// TIA Portal V19 export
FUNCTION_BLOCK "LAF_InterfaceSignalsBool"   // FB52, LAD
TITLE = LAF_InterfaceSignalsBool / Schnittstelle für boolsche Signale
AUTHOR : Siemens Digital Industries
FAMILY : LAF
VERSION : 1.2
// The block cyclically evaluates the status of the configured Boolean signals and transfers the values to the configured data (HMI) interface. The symbolic name of the configured tags will be read once only, triggered by the selection of a signal dataset on the HMI, and will be transferred to the HMI interface as well.  
// The block and the associated WinCC screen are designed for 16 signal datasets with 32 signals each  (“Page 1” through “Page 16”).  The signal dataset can be selected in the WinCC-screen.  
// 
// * The maximum length of the symbol name is limited to 40 characters.  
// 
// For further notes see:  [CallInterfaceSignals](../Function%20Blocks/CallInterfaceSignals.htm)  
// 
// **PLC Data types**  
// * LAF_typeInterfaceSignals  
// + LAF_typeInterfaceSignalsBool  
// 
// **WinCC Screen**  
// {.pageWidth}
// ![Image](LAF_InterfaceSignalsBool/en/image1.PNG)
// 
// **Block call example**  
// {.pageWidth}
// ![Image](LAF_InterfaceSignalsBool/en/image4.PNG)
// View in ladder logic (LAD).  
// 
// **Calling Interface**  
// The block has to be called in the cyclic program in “CallInterfaceSignals”.  
// The block handles 16 Boolean signals. Since one HMI screen can display 32 signals, it is necessary to call the block two times.  
// 
// **Internally used “Extended instructions / blocks“**  
// GetSymbolName
// Die hier aufgeführten Bausteine gehören zum mehrsprachigen Alarm-Bausteinpaket von SICAR in Verbindung mit dem Softwarepaket „ProDiag“.  
// Alle Bausteine besitzt mehrere Input-Parameter „….TriggerX“ an die ein oder mehrere logische Verknüpfungen angelegt werden können. Die Trigger-Eingänge werden mittels ProDiag auf eine Operanden Überwachung überwacht (“Eigenschaften > Überwachung > Allgemein > Überwachungsart: Operand“). Demzufolge sind sie im Fehlerfall auch über den PLC-Code-Viewer auf dem HMI diagnostizierbar.  
// Entsprechend den Überwachungseinstellungen von „ProDiag“ werden die Meldetexte gebildet und erscheinen auf dem HMI in der Meldeanzeige (Bilder: „Meldungen“ / „Alarms“ und „Meldearchiv“ / „Alarms history“). Die Bausteine greifen dazu auf Texte von PLC-Meldetextlisten zu. 
// Eine Meldung kann mehrsprachig ausgeführt werden. Bereits ausgeführte Sprachen sind Englisch und Deutsch; weitere Sprachen sind frei wählbar.  
// Die auf dem HMI angezeigte Sprachvariante wird im Bild „System & Einstellungen“ / “System & Settings“ mit den Buttons der Länderflaggen ausgewählt. Das Bild ist erreichbar, über den Button „System“ (unten rechts im Bild).  
// Ein Bausteinaufruf kann max. 16 Meldungen bearbeiten.  
// 
// WARNING 
// :     Innerhalb des Bausteins wird aufgrund der ProDiag-Überwachung auf PLC-Meldetextliste „GLOBAL_GENERAL_AlarmTextList“ und deren Einträge fest verwiesen. 
// :     ![Icon](_Icon/prohibition.PNG) {.alignLeft} Ändern Sie nicht den Namen dieser PLC-Meldetextliste; der Name wird bei einem Übersetzen im Baustein nicht automatisch nachgeführt!
// :     ![Icon](_Icon/prohibition.PNG) {.alignLeft} Ändern Sie nicht die Reihenfolge der Einträge in der bereits existierenden PLC-Meldetextliste. Diese werden fest referenziert! 
// :     ![Icon](_Icon/information.PNG) {.alignLeft} Sie können stattdessen einen Eintrag in der PLC-Meldetextliste neu hinzufügen.  
// 
// ---
// 
// NOTE
// :     Beachten Sie dabei bitte, dass bei SICAR-Versionsänderungen auch Einträge in den PLC-Meldetextlisten geändert/hinzugefügt werden können, aufgrund dessen es dann zu Doppelbelegungen kommen kann. 
// :     Es ist daher sinnvoll weitere „USER…“-Textliste(n) zu erstellen, losgelöst von den in SICAR bereits existierenden PLC-Meldetextlisten 
// 
// ---
// 
// Es sind folgende Bausteine verfügbar: 
// 
// * LSicar_AlarmOp16_PrD: 		16 Operanden Alarme (rote Hintergrundfarbe im Alarm-Bild)
// * LSicar_WarnOp16_PrD: 		16 Operanden Warnungen (orange Hintergrundfarbe im Alarm-Bild) 
// * LSicar_InfoOp16_PrD: 		16 Operanden Informationen (blaue Hintergrundfarbe im Alarm-Bild) 
// *  LSicar_AlarmOpFsafe8_PrD: 		8 Operanden F-Alarme (gelbe Hintergrundfarbe im Alarm-Bild) 
// 
// **Überwachungsart**  
// 
// ![Image](LSicar_AlarmOp16_PrD/de/image1.PNG) 
// 
// Der Text für die Überwachungsart „Fehlermeldung“ ist in den  Überwachungseinstellungen „Allgemein > Überwachungsart > Eigenschaften“ mit -Op- angegeben und bei der Projektierung der „Meldetexte > FB-Parameter“ im Meldetext konfiguriert.  
// 
// **_AlarmOp16_PrD**  
// In den ProDiag-Überwachungseinstellungen ist die Kategorie: „Alarm“ definiert und wird für alle Inputs verwendet. Dieser Kategorie ist die Meldeklasse „ Alarm_ProDiag“ zugeordnet. Auf dem HMI ist dieser Meldeklasse unter „HMI-Meldungen > Lasche ‚Meldeklasse‘“ die Hintergrundfarbe Rot zugeordnet mit dem Anzeigename „Alarm“. Somit erscheinen Meldungen im Alarm-Bild wie folgt (Beispiel):  
// 
// ![Image](LSicar_AlarmOp16_PrD/de/image2.PNG)  
// 
// Zudem werden die Alarme auf eine Statische Variable „HMI_Alarm“ kopiert. Diese kann dazu benutzt werden um ein HMI-Variable zu generieren und -somit auf dem HMI- die Signale zu Animationszwecken zu nutzen.  
// 
// **_WarnOp16_PrD**  
// In den ProDiag-Überwachungseinstellungen ist die Kategorie: „Warn“ definiert und wird für alle Inputs verwendet. Dieser Kategorie ist die Meldeklasse „ Warning_ProDiag“ zugeordnet. Auf dem HMI ist dieser Meldeklasse unter „HMI-Meldungen > Lasche ‚Meldeklasse‘“ die Hintergrundfarbe Orange zugeordnet mit dem Anzeigename „Warn“. Somit erscheinen Meldungen im Alarm-Bild wie folgt (Beispiel):  
// 
// ![Image](LSicar_AlarmOp16_PrD/de/image3.PNG)
// 
// The warnings are also copied to a static tag “HMI_Warn”. This can be used to generate a HMI tag, e.g. to use the signals for animations on the HMI.  
// 
// **_InfoOp16_PrD**  
// In den ProDiag-Überwachungseinstellungen ist die Kategorie: „Info“ definiert und wird für alle Inputs verwendet. Dieser Kategorie ist die Meldeklasse „ Information_ProDiag“ zugeordnet. Auf dem HMI ist dieser Meldeklasse unter „HMI-Meldungen > Lasche ‚Meldeklasse‘“ die Hintergrundfarbe Blau zugeordnet mit dem Anzeigename „Info“. Somit erscheinen Meldungen im Alarm-Bild wie folgt (Beispiel):  
// 
// ![Image](LSicar_AlarmOp16_PrD/de/image4.PNG)
// 
// Zudem werden die Warnungen auf eine Statische Variable „HMI_Warn“ kopiert. Diese kann dazu benutzt werden um ein HMI-Variable zu generieren und -somit auf dem HMI- die Signale zu Animationszwecken zu nutzen.  
// 
// **_AlarmOpFsafe8_PrD**  
// In den ProDiag-Überwachungseinstellungen ist die Kategorie: „F-Alarm“ definiert und wird für alle Inputs verwendet. Dieser Kategorie ist die Meldeklasse „F-Alarm_ProDiag“ zugeordnet. Auf dem HMI ist dieser Meldeklasse unter „HMI-Meldungen > Lasche ‚Meldeklasse‘“ die Hintergrundfarbe Gelb zugeordnet mit dem Anzeigename „F-Alarm“. Somit erscheinen Meldungen im Alarm-Bild wie folgt (Beispiel):  
// 
// ![Image](LSicar_AlarmOp16_PrD/de/image5.PNG)
// 
// Zudem werden die Meldungen auf Statische Variablen „HMI_Alarm…“ kopiert. Diese können dazu benutzt werden um HMI-Variablen zu generieren und -somit auf dem HMI- die Signale zu Animationszwecken zu nutzen.  
// 
//  
// #### ProDiag-Meldung in 3 Schritten 
// 
// {.pageWidth}
// ![Image](LSicar_AlarmOp16_PrD/de/image6.PNG)
// 
// **1) Legen Sie eine PLC-Meldetextliste an**
// 1. Öffnen Sie dazu (im Projektbaum) „PLC-Meldetextlisten“ und vergeben Sie einen Namen, hier „Demo_Alarm_PD“.  
// 2. Geben Sie den jeweiligen Meldetext in die Spalte „Eintrag“ ein.
// 	- Achten Sie darauf das die Spalten „Bereich von“ und „Bereich bis“ den gleichen Wert haben.  
// 	- Beginnen Sie mit dem Wert 1.  
// 	- Der Eintrag 1 entspricht dem FB-Parameter „…_trigger1“,  
// 	- Eintrag 2 entspricht FB-Parameter „…_trigger2“, usw.  
// 
// 3. Projektieren Sie die Einträge in den gewünschten Sprachen (hier: Deutsch und Englisch). 
// 
// {.pageWidth}
// ![Image](LSicar_AlarmOp16_PrD/de/image7.PNG)
// 
// **2) Eintrag in „GLOBAL_GENERAL_AlarmTextList“**  
// 1. Öffnen Sie die Textliste „GLOBAL_GENERAL_AlarmTextList“.  
// 2. Tragen Sie den Namen der Textliste, die Sie erzeugt haben, als einen neuen Eintrag ein. Fügen Sie sie dabei als neuen Eintrag hinzu (hier Eintrag 25). Geben Sie dabei den Namen der Textliste als Begleitwert ein mit @4%t#<Namen>@.  
// 3. Projektieren Sie dies in allen gewünschten Sprachen.  
//  
// {.pageWidth}
// ![Image](LSicar_AlarmOp16_PrD/de/image8.PNG)
//  
// **3 Rufen Sie den Alarm-Baustein auf**   
// 1. Geben Sie beim Parameter „plantIdentifier“ einen zusätzlichen Text an. Dieser erscheint ebenso im Meldetext.  
// 2. Beim Parameter „globalAlarmTextlistItem“ geben Sie den Wert des Eintrags an „Bereich von“ / „Bereich bis“, unter dem Ihre Textliste in der „GLOBAL_GENERAL_AlarmTextList“ eingetragen ist, hier 25; damit verweisen Sie auf Ihre PLC-Meldetextliste.  
// 3. Versorgen Sie die Trigger-Eingänge.  
// 
// {.pageWidth}
// ![Image](LSicar_AlarmOp16_PrD/de/image9.PNG)
// 
// **Ergebnise:**  
// Wechselt der Trigger-Eingang auf „1“-Signal, so erscheint die Meldung im Alarm-Bild (entsprechend der ProDiag-Konfiguration) und es kann in den PLC-Code-Viewer verzweigt werden.  
// 
// {.pageWidth}
// ![Image](LSicar_AlarmOp16_PrD/de/image10.PNG)
// 
// 
// **Beispielaufruf**  
// Abbildung in Kontaktplan (KOP), ohne Parameterbeschaltung.  
// Ein lauffähiger Programm-Aufruf hierzu ist im „SICAR-StartUp“-Projekt enthalten.  
// 
// **Aufrufschnittstelle**
// Der Baustein wird im zyklischen Programm aufgerufen.
// stored: Access Published, IsIECCheckEnabled true, MemoryReserve 100, SetENOAutomatically true
   VAR_INPUT
      signal00 { ExternalAccessible := 'False'; ExternalVisible := 'False'; ExternalWritable := 'False'} : Bool;   // Boolesches Signal (01) dessen Status und symbolischer Name am HMI dargestellt werden soll. Hinweis: Der symbolische Namen wird mit max. 32 Zeichen darge-stellt. / Boolean signal (number 01) to be displayed on the HMI with status and symbolic name.
      signal01 { ExternalAccessible := 'False'; ExternalVisible := 'False'; ExternalWritable := 'False'} : Bool;   // Analoge Parametrierung wie bei Input „signal01“ / Similar configuration as for “signal01“
      signal02 { ExternalAccessible := 'False'; ExternalVisible := 'False'; ExternalWritable := 'False'} : Bool;   // Analoge Parametrierung wie bei Input „signal01“ / Similar configuration as for “signal01“
      signal03 { ExternalAccessible := 'False'; ExternalVisible := 'False'; ExternalWritable := 'False'} : Bool;   // Analoge Parametrierung wie bei Input „signal01“ / Similar configuration as for “signal01“
      signal04 { ExternalAccessible := 'False'; ExternalVisible := 'False'; ExternalWritable := 'False'} : Bool;   // Analoge Parametrierung wie bei Input „signal01“ / Similar configuration as for “signal01“
      signal05 { ExternalAccessible := 'False'; ExternalVisible := 'False'; ExternalWritable := 'False'} : Bool;   // Analoge Parametrierung wie bei Input „signal01“ / Similar configuration as for “signal01“
      signal06 { ExternalAccessible := 'False'; ExternalVisible := 'False'; ExternalWritable := 'False'} : Bool;   // Analoge Parametrierung wie bei Input „signal01“ / Similar configuration as for “signal01“
      signal07 { ExternalAccessible := 'False'; ExternalVisible := 'False'; ExternalWritable := 'False'} : Bool;   // Analoge Parametrierung wie bei Input „signal01“ / Similar configuration as for “signal01“
      signal08 { ExternalAccessible := 'False'; ExternalVisible := 'False'; ExternalWritable := 'False'} : Bool;   // Analoge Parametrierung wie bei Input „signal01“ / Similar configuration as for “signal01“
      signal09 { ExternalAccessible := 'False'; ExternalVisible := 'False'; ExternalWritable := 'False'} : Bool;   // Analoge Parametrierung wie bei Input „signal01“ / Similar configuration as for “signal01“
      signal10 { ExternalAccessible := 'False'; ExternalVisible := 'False'; ExternalWritable := 'False'} : Bool;   // Analoge Parametrierung wie bei Input „signal01“ / Similar configuration as for “signal01“
      signal11 { ExternalAccessible := 'False'; ExternalVisible := 'False'; ExternalWritable := 'False'} : Bool;   // Analoge Parametrierung wie bei Input „signal01“ / Similar configuration as for “signal01“
      signal12 { ExternalAccessible := 'False'; ExternalVisible := 'False'; ExternalWritable := 'False'} : Bool;   // Analoge Parametrierung wie bei Input „signal01“ / Similar configuration as for “signal01“
      signal13 { ExternalAccessible := 'False'; ExternalVisible := 'False'; ExternalWritable := 'False'} : Bool;   // Analoge Parametrierung wie bei Input „signal01“ / Similar configuration as for “signal01“
      signal14 { ExternalAccessible := 'False'; ExternalVisible := 'False'; ExternalWritable := 'False'} : Bool;   // Analoge Parametrierung wie bei Input „signal01“ / Similar configuration as for “signal01“
      signal15 { ExternalAccessible := 'False'; ExternalVisible := 'False'; ExternalWritable := 'False'} : Bool;   // Analoge Parametrierung wie bei Input „signal01“ / Similar configuration as for “signal01“
   END_VAR
   VAR_IN_OUT
      interfaceSignals : "LAF_typeInterfaceSignalsBool";   // Im FB “CallInterfaceSignals“ existiert die Struktur „statInterfaceSignalsHmi“ (Array[0..16] of „typeInterfaceSignals-Hmi“). In jeder Struktur existieren die Elemente: - „valueSymboLeft“ und - „valueSymbolRight“mit dem Datentyp "_typeInterfaceSignalsBool"“. Die Nummer des Arrays entspricht dem Signaldatensatz: - Array [1]: Signaldatensatz 1 - Array [2]: Signaldatensatz 2 - usw.Array Index [0] ist nicht zulässig.Zuweisung der entsprechenden Variablen, wie nachfolgend beispiel-haft dargestellt. Der rechte Aufruf entspricht den 16 Signalen auf der rechten Seite des Bildes, der linke Aufruf der linken Seite. / “CallInterfaceSignals“ contains the structure “statInterfaceSignalsHmi“ (Array[0..16] of „typeInterfaceSignalsHmi“). Within each structure there are the two elements: “valueSymbolLeft” and “valueSymbolRight” of the data type “LAF_typeInterfaceSignalsBool“. The number of the array correlates with the number of the signal data-set: Array [1]: Signal data set 1 and Array [2]: Signal data set 2 etc. Array index [0] is not permitted.
   END_VAR
   VAR_TEMP
      tempDummyBool : Bool;   // Dummy
   END_VAR
BEGIN

REGION Network 1: Header Info / Änderungshistorie
   // SIEMENS AG / (c)Copyright 2024
   // ------------------------------------------------------------------------------
   // Title:            LAF_InterfaceSignalsBool
   // Comment/Function: The block cyclically evaluates the status of the configured Boolean signals and transfers the values to the configured data (HMI) interface.
   // Library/Family:           Library of Automation Framework
   // Author:             Siemens Digital Industry
   // Tested with:    S7-PLCSIM Advanced 6.0
   // Engineering:   TIA Portal V19
   // Restrictions:     ---
   // Requirements: ---
   // ------------------------------------------------------------------------------
   // Change log table:
   // Version | Date | Expert in charge | Changes applied
   // -------|---------|-------------|--------------------------------------------
   // 01.02.00 | 30.09.2024 | SIMATIC Systems Support | First released version
   // Die Änderungshistorie wird nur in englischer Editiersprache geführt.
END_REGION

REGION Network 2: Description / Beschreibung
   // **Operation mode Automatic / Manual**  
   // The block is independent of the operation modes and is not assigned to any operation mode area.  
   // 
   // **Alarms**  
   // The block does not generate alarms.  
   // 
   // #### PLC Data types  
   // 
   // The PLC data types are used to structure the data in FB “CallInterfaceSignals“.  
   // 
   // * [LAF_typeInterfaceSignals](../Library%20Types/LAF_typeInterfaceSignals.htm)  
   // * [LAF_typeInterfaceSignalsBool](../Library%20Types/LAF_typeInterfaceSignalsBool.htm)  
   // 
   // #### WinCC-Screen objects 
   // 
   // **WinCC Diagnostic screen**  
   // The screen is located in the project in HMI part under screens -> 09_Diagnostics.  
   // The selection of the interface signal screens is done via the navigation screens which are stored in 00_Screenlayout -> ThirdMenus.  
   // The status is animated in terms of color. Status TRUE = green, Status FALSE = gray.  
   // 
   // **Example**  
   // The Boolean status of the system and clock bit memories are displayed in the screen. The corresponding dataset can be selected via the third navigation bar on the left side of the screen. A headline text can be 
   // entered for each column in the PLC – InstInterfaceSignals DB -> statInterfaceSignalsHmi.  
   // 
   // {.pageWidth}
   // ![Image](LAF_InterfaceSignalsBool/en/image3.PNG)
   // 
   //  
   // #### Further information 
   // 
   // #### Update info 
   // 
   // #### Further documentation  
   // * See [CallInterfaceSignals](../Function%20Blocks/CallInterfaceSignals.htm)
   // **Betriebsart Automatik/Hand**  
   // Der Baustein ist Betriebsarten unabhängig und wird daher keinem Betriebsartenbereich zugewiesen.  
   // 
   // **Alarme**  
   // Der Baustein löst keine eigenen Alarme aus.  
   // 
   // **Beispiel** 
   // 1)	Der Baustein wird aufgerufen mit globalAlarmTextlistItem:= 1. Damit wird auf die PLC-Meldetextliste „OPMode01_Alarm_PD“ verwiesen. Der Input „alarmTrigger1“ zeigt auf den 1. Eintrag in dieser PLC-Meldetextliste.  
   // 2)	Die Überwachung an „alarmTrigger1“ soll auf „0“-Signal (False) überwacht werden; daher die NOT-Verknüpfung.  
   // 
   // {.pageWidth}
   // ![Image](LSicar_AlarmOp16_PrD/de/image10.PNG)
   // 
   // 3)	Die Meldung wird im Alarmbild dargestellt  
   // 4)	und kann im PLC-Viewer beobachtet werden.  
   // 
   // {.pageWidth}
   // ![Image](LSicar_AlarmOp16_PrD/de/image11.PNG)
   // 
   // #### Weitere Dokumente
   // 
   // ![Icon](_Icon/reference.PNG)  
   // 
   // - ProDiag Einstellungen in SICAR: ..\SICAR_Global\SICAR_ProDiag_Settings.pdf  
   // - SICAR PLC Meldetextlisten: ..\SICAR_Global\SICAR_PLC_AlarmTextLists.pdf
END_REGION

REGION Network 3: Update boolean value / Aktualisieren der boolschen Werte
   // Cyclic update of the boolean signal, if the screen is loaded / Wert des Boolschen Signals wird zyklisch aktualisiert, wenn das Bild aufgerufen ist
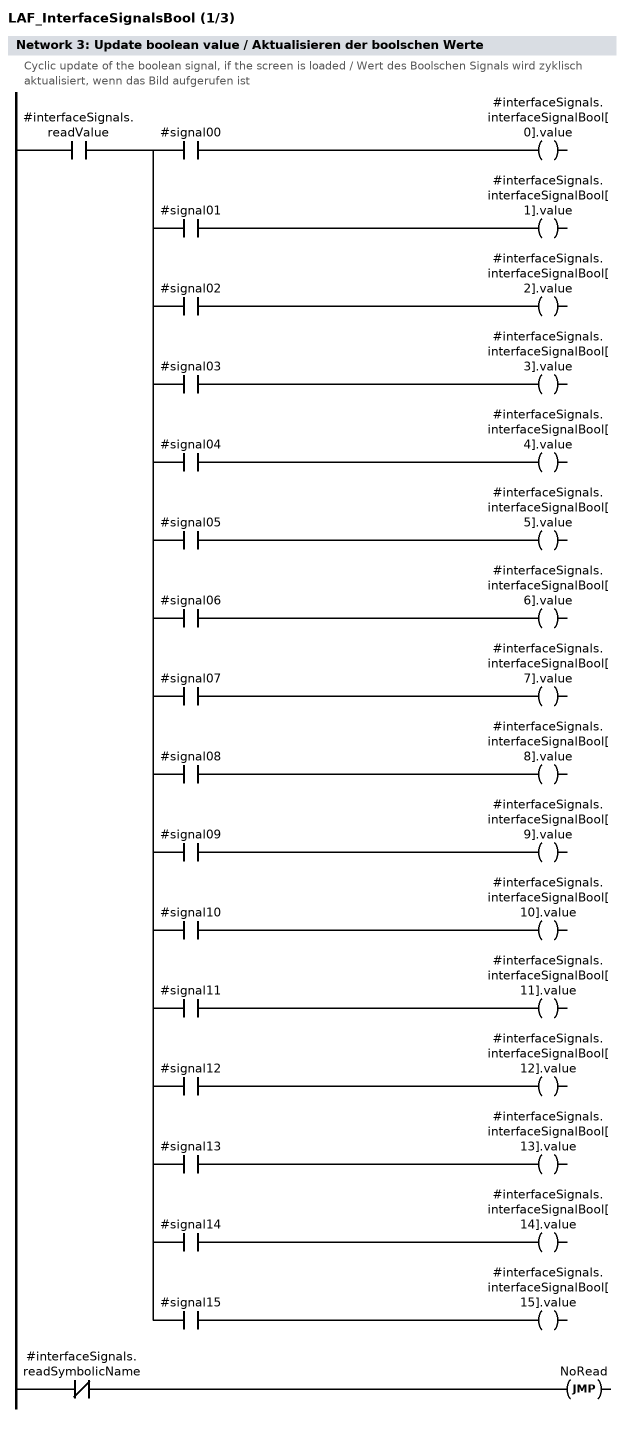
   RUNG wire#powerrail
      Contact( #interfaceSignals.readValue )
      wire#w1
      Contact( #signal00 )
      Coil( #interfaceSignals.interfaceSignalBool[0].value )
   END_RUNG
   RUNG wire#w1
      Contact( #signal01 )
      Coil( #interfaceSignals.interfaceSignalBool[1].value )
   END_RUNG
   RUNG wire#w1
      Contact( #signal02 )
      Coil( #interfaceSignals.interfaceSignalBool[2].value )
   END_RUNG
   RUNG wire#w1
      Contact( #signal03 )
      Coil( #interfaceSignals.interfaceSignalBool[3].value )
   END_RUNG
   RUNG wire#w1
      Contact( #signal04 )
      Coil( #interfaceSignals.interfaceSignalBool[4].value )
   END_RUNG
   RUNG wire#w1
      Contact( #signal05 )
      Coil( #interfaceSignals.interfaceSignalBool[5].value )
   END_RUNG
   RUNG wire#w1
      Contact( #signal06 )
      Coil( #interfaceSignals.interfaceSignalBool[6].value )
   END_RUNG
   RUNG wire#w1
      Contact( #signal07 )
      Coil( #interfaceSignals.interfaceSignalBool[7].value )
   END_RUNG
   RUNG wire#w1
      Contact( #signal08 )
      Coil( #interfaceSignals.interfaceSignalBool[8].value )
   END_RUNG
   RUNG wire#w1
      Contact( #signal09 )
      Coil( #interfaceSignals.interfaceSignalBool[9].value )
   END_RUNG
   RUNG wire#w1
      Contact( #signal10 )
      Coil( #interfaceSignals.interfaceSignalBool[10].value )
   END_RUNG
   RUNG wire#w1
      Contact( #signal11 )
      Coil( #interfaceSignals.interfaceSignalBool[11].value )
   END_RUNG
   RUNG wire#w1
      Contact( #signal12 )
      Coil( #interfaceSignals.interfaceSignalBool[12].value )
   END_RUNG
   RUNG wire#w1
      Contact( #signal13 )
      Coil( #interfaceSignals.interfaceSignalBool[13].value )
   END_RUNG
   RUNG wire#w1
      Contact( #signal14 )
      Coil( #interfaceSignals.interfaceSignalBool[14].value )
   END_RUNG
   RUNG wire#w1
      Contact( #signal15 )
      Coil( #interfaceSignals.interfaceSignalBool[15].value )
   END_RUNG
   RUNG wire#powerrail
      I_Contact( #interfaceSignals.readSymbolicName )
      JumpCoil( NoRead )
   END_RUNG
   // the same network as SCL:
   #interfaceSignals.interfaceSignalBool[0].value := #interfaceSignals.readValue AND #signal00;
   #interfaceSignals.interfaceSignalBool[1].value := #interfaceSignals.readValue AND #signal01;
   #interfaceSignals.interfaceSignalBool[2].value := #interfaceSignals.readValue AND #signal02;
   #interfaceSignals.interfaceSignalBool[3].value := #interfaceSignals.readValue AND #signal03;
   #interfaceSignals.interfaceSignalBool[4].value := #interfaceSignals.readValue AND #signal04;
   #interfaceSignals.interfaceSignalBool[5].value := #interfaceSignals.readValue AND #signal05;
   #interfaceSignals.interfaceSignalBool[6].value := #interfaceSignals.readValue AND #signal06;
   #interfaceSignals.interfaceSignalBool[7].value := #interfaceSignals.readValue AND #signal07;
   #interfaceSignals.interfaceSignalBool[8].value := #interfaceSignals.readValue AND #signal08;
   #interfaceSignals.interfaceSignalBool[9].value := #interfaceSignals.readValue AND #signal09;
   #interfaceSignals.interfaceSignalBool[10].value := #interfaceSignals.readValue AND #signal10;
   #interfaceSignals.interfaceSignalBool[11].value := #interfaceSignals.readValue AND #signal11;
   #interfaceSignals.interfaceSignalBool[12].value := #interfaceSignals.readValue AND #signal12;
   #interfaceSignals.interfaceSignalBool[13].value := #interfaceSignals.readValue AND #signal13;
   #interfaceSignals.interfaceSignalBool[14].value := #interfaceSignals.readValue AND #signal14;
   #interfaceSignals.interfaceSignalBool[15].value := #interfaceSignals.readValue AND #signal15;
   IF NOT #interfaceSignals.readSymbolicName THEN GOTO NoRead; END_IF;
END_REGION

REGION Network 4: Read symbolic name / Symbolischen Namen lesen
   // Symbolic name of boolean signals will be actualized once only after screen active / Symbolischer Name des Boolschen Signals wird einmalig aktualisiert, wenn das Bild aufgerufen ist
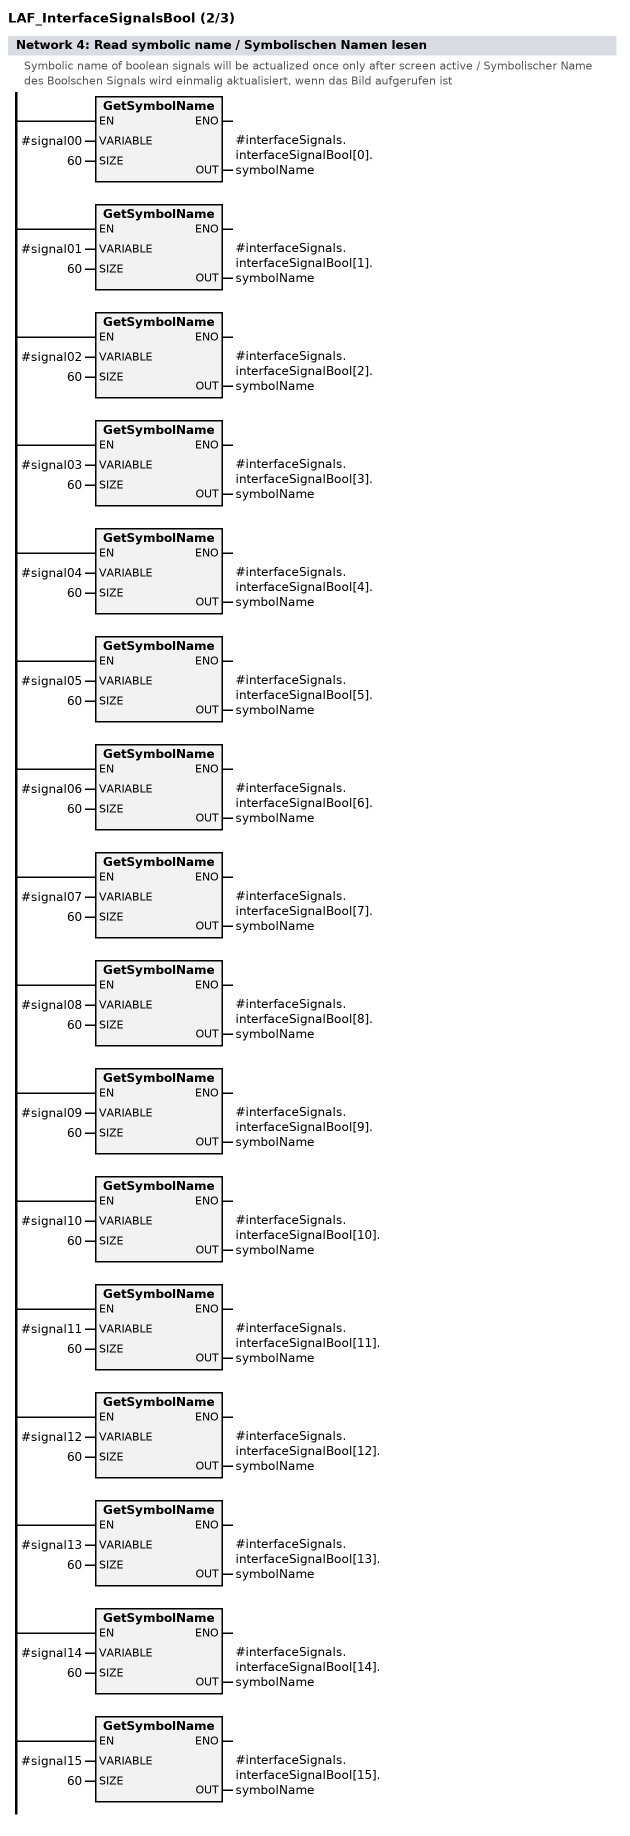
   RUNG wire#powerrail
      GetSymbolName(variable := #signal00, size := 60, OUT => #interfaceSignals.interfaceSignalBool[0].symbolName)
   END_RUNG
   RUNG wire#powerrail
      GetSymbolName(variable := #signal01, size := 60, OUT => #interfaceSignals.interfaceSignalBool[1].symbolName)
   END_RUNG
   RUNG wire#powerrail
      GetSymbolName(variable := #signal02, size := 60, OUT => #interfaceSignals.interfaceSignalBool[2].symbolName)
   END_RUNG
   RUNG wire#powerrail
      GetSymbolName(variable := #signal03, size := 60, OUT => #interfaceSignals.interfaceSignalBool[3].symbolName)
   END_RUNG
   RUNG wire#powerrail
      GetSymbolName(variable := #signal04, size := 60, OUT => #interfaceSignals.interfaceSignalBool[4].symbolName)
   END_RUNG
   RUNG wire#powerrail
      GetSymbolName(variable := #signal05, size := 60, OUT => #interfaceSignals.interfaceSignalBool[5].symbolName)
   END_RUNG
   RUNG wire#powerrail
      GetSymbolName(variable := #signal06, size := 60, OUT => #interfaceSignals.interfaceSignalBool[6].symbolName)
   END_RUNG
   RUNG wire#powerrail
      GetSymbolName(variable := #signal07, size := 60, OUT => #interfaceSignals.interfaceSignalBool[7].symbolName)
   END_RUNG
   RUNG wire#powerrail
      GetSymbolName(variable := #signal08, size := 60, OUT => #interfaceSignals.interfaceSignalBool[8].symbolName)
   END_RUNG
   RUNG wire#powerrail
      GetSymbolName(variable := #signal09, size := 60, OUT => #interfaceSignals.interfaceSignalBool[9].symbolName)
   END_RUNG
   RUNG wire#powerrail
      GetSymbolName(variable := #signal10, size := 60, OUT => #interfaceSignals.interfaceSignalBool[10].symbolName)
   END_RUNG
   RUNG wire#powerrail
      GetSymbolName(variable := #signal11, size := 60, OUT => #interfaceSignals.interfaceSignalBool[11].symbolName)
   END_RUNG
   RUNG wire#powerrail
      GetSymbolName(variable := #signal12, size := 60, OUT => #interfaceSignals.interfaceSignalBool[12].symbolName)
   END_RUNG
   RUNG wire#powerrail
      GetSymbolName(variable := #signal13, size := 60, OUT => #interfaceSignals.interfaceSignalBool[13].symbolName)
   END_RUNG
   RUNG wire#powerrail
      GetSymbolName(variable := #signal14, size := 60, OUT => #interfaceSignals.interfaceSignalBool[14].symbolName)
   END_RUNG
   RUNG wire#powerrail
      GetSymbolName(variable := #signal15, size := 60, OUT => #interfaceSignals.interfaceSignalBool[15].symbolName)
   END_RUNG
   // the same network as SCL:
   GetSymbolName(variable := #signal00, size := 60, OUT => #interfaceSignals.interfaceSignalBool[0].symbolName);
   GetSymbolName(variable := #signal01, size := 60, OUT => #interfaceSignals.interfaceSignalBool[1].symbolName);
   GetSymbolName(variable := #signal02, size := 60, OUT => #interfaceSignals.interfaceSignalBool[2].symbolName);
   GetSymbolName(variable := #signal03, size := 60, OUT => #interfaceSignals.interfaceSignalBool[3].symbolName);
   GetSymbolName(variable := #signal04, size := 60, OUT => #interfaceSignals.interfaceSignalBool[4].symbolName);
   GetSymbolName(variable := #signal05, size := 60, OUT => #interfaceSignals.interfaceSignalBool[5].symbolName);
   GetSymbolName(variable := #signal06, size := 60, OUT => #interfaceSignals.interfaceSignalBool[6].symbolName);
   GetSymbolName(variable := #signal07, size := 60, OUT => #interfaceSignals.interfaceSignalBool[7].symbolName);
   GetSymbolName(variable := #signal08, size := 60, OUT => #interfaceSignals.interfaceSignalBool[8].symbolName);
   GetSymbolName(variable := #signal09, size := 60, OUT => #interfaceSignals.interfaceSignalBool[9].symbolName);
   GetSymbolName(variable := #signal10, size := 60, OUT => #interfaceSignals.interfaceSignalBool[10].symbolName);
   GetSymbolName(variable := #signal11, size := 60, OUT => #interfaceSignals.interfaceSignalBool[11].symbolName);
   GetSymbolName(variable := #signal12, size := 60, OUT => #interfaceSignals.interfaceSignalBool[12].symbolName);
   GetSymbolName(variable := #signal13, size := 60, OUT => #interfaceSignals.interfaceSignalBool[13].symbolName);
   GetSymbolName(variable := #signal14, size := 60, OUT => #interfaceSignals.interfaceSignalBool[14].symbolName);
   GetSymbolName(variable := #signal15, size := 60, OUT => #interfaceSignals.interfaceSignalBool[15].symbolName);
END_REGION

REGION Network 5: End of block / Ende des Bausteins
   // Jump lable "NoRead" to read the symbolic name only once / Sprungmarke "NoRead" um den symbolischen Namen nur einmal zu lesen
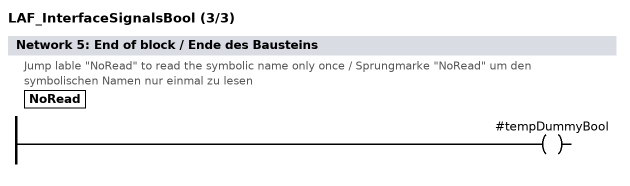
   Label( NoRead )
   RUNG wire#powerrail
      Coil( #tempDummyBool )
   END_RUNG
   // the same network as SCL:
   NoRead:
   #tempDummyBool := TRUE;
END_REGION
END_FUNCTION_BLOCK
